// LS Electric XG5000 project: 123
// PLC NewPLC
// module base 0 slot 0: 입출력 모듈:XBC-DR32H (DC 24V 입력, 릴레이 출력 32점)

PROGRAM NewProgram (task: 스캔 프로그램)

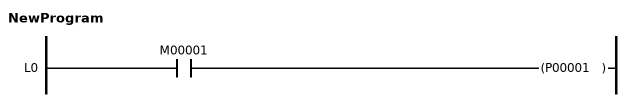
; L0
LOAD      M00001
OUT       P00001

VARIABLES AND COMMENTS (devices not used above)
M00000	BIT	PB1